TYPE EcMasterInputs :
STRUCT
	SlaveCount : UINT;
	DevState : UINT;
END_STRUCT
END_TYPE

(* stored: Version 1.1.0.1, ProductVersion 3.1.4024.11
   DUT EcMasterInputs: Id {6d14eb69-f187-42a0-a00b-1e0fd8ba899c} *)
